(* IEC 61131-3 sources: dynamics/src/Controllers, 3 files *)

(* ---- IDynamicController.st ---- *)
NAMESPACE Simatic.Ax.Dynamics
    INTERFACE IDynamicController

        METHOD Next : LREAL
            VAR_INPUT
                value : LREAL;
                input : LREAL;
            END_VAR
        END_METHOD

    END_INTERFACE
END_NAMESPACE

(* ---- BangBangController.st ---- *)
NAMESPACE Simatic.Ax.Dynamics
    CLASS BangBangController EXTENDS Controller

        VAR PUBLIC
            hysteresis : LREAL;
        END_VAR
        VAR PRIVATE
            _output : BOOL;
            _heatingMode : BOOL;
        END_VAR

        // Get Output
        METHOD PUBLIC GetOutput : BOOL
            GetOutput := _output;
        END_METHOD
        // Set Output
        METHOD PUBLIC SetOutput
            VAR_INPUT
                newOutput : BOOL;
            END_VAR
            _output := newOutput;
        END_METHOD

        // Get Mode
        METHOD PUBLIC IsHeatingModeEnabled : BOOL
            IsHeatingModeEnabled := _heatingMode;
        END_METHOD
        METHOD PUBLIC IsCoolingModeEnabled : BOOL
            IsCoolingModeEnabled := NOT _heatingMode;
        END_METHOD
        // Set Mode
        METHOD PUBLIC EnableHeatingMode
            _heatingMode := TRUE;
        END_METHOD
        METHOD PUBLIC EnableCoolingMode
            _heatingMode := FALSE;
        END_METHOD

        METHOD PUBLIC Next : BOOL
            VAR_INPUT
                value : LREAL;
            END_VAR
            IF      value < this.GetInput() - hysteresis * 0.5 THEN
                _output := _heatingMode;
            ELSIF   value > this.GetInput() + hysteresis * 0.5  THEN
                _output := NOT _heatingMode;
            END_IF;
            Next := _output;
        END_METHOD

        METHOD PUBLIC Next : BOOL
            VAR_INPUT
                value : LREAL;
                input : LREAL;
            END_VAR
            this.SetInput(input);
            Next := this.Next(value);
        END_METHOD

    END_CLASS
END_NAMESPACE

(* ---- PT1_DeadbeatController.st ---- *)
USING System.Math;
NAMESPACE Simatic.Ax.Dynamics
    CLASS PT1_DeadbeatController EXTENDS Controller IMPLEMENTS IDynamicController

        VAR PROTECTED
            _expTT : LREAL;
            _k : LREAL;
        END_VAR

        // Get K
        METHOD PUBLIC GetK : LREAL
            GetK := _k;
        END_METHOD
        // Set K
        METHOD PUBLIC SetK
            VAR_INPUT
                k : LREAL;
            END_VAR
            _k := k;
        END_METHOD

        // Set T0
        METHOD PUBLIC SetPeriods
            VAR_INPUT
                elapsedTime : LREAL;
                t0 : LREAL;
            END_VAR
            _expTT := Exp(elapsedTime / t0);
        END_METHOD

        METHOD PUBLIC Next : LREAL
            VAR_INPUT
                value : LREAL;
            END_VAR
            Next := (THIS.GetInput() * _expTT - value) / (_expTT - 1) / _k;
        END_METHOD

        METHOD PUBLIC Next : LREAL
            VAR_INPUT
                value : LREAL;
                input : LREAL;
            END_VAR
            THIS.SetInput(input);
            Next := THIS.Next(value);
        END_METHOD

    END_CLASS
END_NAMESPACE
